TYPE stBH0KPL_Line EXTENDS stPIM_LineEventsModule :
STRUCT

	{attribute 'OPC.UA.DA' := '1'}
	stStation_BH0KPL01 : stPIM_StationEventsModule_3_Machine;
END_STRUCT
END_TYPE

(* stored: Version 1.1.0.1, ProductVersion 3.1.4024.15
   DUT stBH0KPL_Line: Id {1be6c9a7-35c9-4ec6-92e1-23d4092f81f7} *)
